Yaskawa INFORM job: SYS_FILTERS_STOP.JBI

/JOB
//NAME SYS_FILTERS_STOP
//POS
///NPOS 0,0,0,0,0,0
//INST
///DATE 2021/12/03 12:01
///ATTR SC,RW
///GROUP1 RB1
NOP
DOUT OT#(20) OFF
DOUT OT#(21) OFF
END
